(*
Integrates the input error signal with back-calculation anti-windup.

Extends :class:`FB_Integrator` by accepting an external comparator input,
typically the :attr:`~FB_Clamp.Residual` of an :class:`FB_Clamp` block, to
unwind the integrator gradually when the output is saturated. The residual is
scaled by ``1 / Tt`` and subtracted from the integrator input each cycle.

A typical wiring pattern:

.. code-block:: pascal

   fbI.Input           := fbP.Output; // Standard form. Use fError for parallel form.
   fbI.ComparatorInput := fbClamp.Residual;
   fbI.Run();
   fbClamp.Input := fbP.Output + fbI.Output + fbD.Output;
   fbClamp.Run();

.. note::
   Set :attr:`Maximum` before :attr:`Minimum` to ensure the clamp guard applies
   correctly.

   Use ``FB_init`` to set :attr:`tTn` and :attr:`tTt` at declaration time.
*)
{attribute 'no_assign'}
{attribute 'enable_dynamic_creation'}
{attribute 'no_explicit_call' := 'direct call for this function block is not allowed'}
FUNCTION_BLOCK FINAL FB_TrackingIntegrator EXTENDS FB_Integrator
VAR
	_fComparatorInput  : LREAL; // External residual signal for back-calculation anti-windup.
	_tTt 			   : LTIME; // Tracking time constant (Tt). Controls how quickly the integrator unwinds.
END_VAR

(*
Gets or sets the comparator input.

This is typically the :attr:`~FB_Clamp.Residual` of an :class:`FB_Clamp` block
placed after the PID summation, passed directly without negation. The block
subtracts the scaled residual from the integrator input internally to unwind
the integrator when the output is saturated.

A positive value indicates the unsaturated sum exceeded the clamp maximum.
A negative value indicates it fell below the clamp minimum.
*)
PROPERTY ComparatorInput : LREAL
GET
ComparatorInput := THIS^._fComparatorInput;
END_GET
SET
THIS^._fComparatorInput := ComparatorInput;
END_SET
END_PROPERTY

METHOD FB_init : BOOL
VAR_INPUT
	bInitRetains : BOOL;  // if TRUE, the retain variables are initialized (warm start / cold start)
	bInCopyCode  : BOOL;  // if TRUE, the instance afterwards gets moved into the copy code (online change)
	tTn          : LTIME; // Integral action time. LTIME#0 disables integration.
	tTt 		 : LTIME; // Tracking time constant (Tt). A typical starting value is SQRT(Tn * Td).
END_VAR
THIS^._tTt := tTt;
END_METHOD

(*
Advances the tracking integrator by one time step.

.. note::
   Must be called once per cycle on a single PLC task. If :attr:`Tn` is
   ``LTIME#0`` the output is set to zero. If :attr:`Tt` is ``LTIME#0``
   the back-calculation correction is disabled.
*)
METHOD Run
VAR_INST
	{attribute 'hide'}
	bInit       : BOOL := TRUE;
	{attribute 'hide'}
	fT          : LREAL;
	{attribute 'hide'}
	fbTaskCycle : FsCommon.FB_PlcTaskCycleChangeDetector(0);
END_VAR
VAR
	fKi         : LREAL;
	fTt         : LREAL;
	fWindupBack : LREAL;
END_VAR
IF bInit THEN
	fT := TO_LREAL(FsCommon.F_GetCurrentTaskCycleTime()) / TO_LREAL(LTIME#1S);
	RETURN(bInit := fT <= 0);
	fbTaskCycle.TaskIndex := FsCommon.F_GetCurrentTaskIndex();
END_IF

RETURN(NOT fbTaskCycle.HasChanged);

THIS^._fMaximum := MAX(THIS^._fMinimum, THIS^._fMaximum);
THIS^._fMinimum := MIN(THIS^._fMinimum, THIS^._fMaximum);

IF FsCommon.F_ResetOnTrue(THIS^._bSync) THEN
	THIS^._fOutput := LIMIT(THIS^._fMinimum, THIS^._fSync, THIS^._fMaximum);
END_IF

IF THIS^._tTn = LTIME#0S THEN
	THIS^._fOutput := 0;
	RETURN;
END_IF

fKi := 1.0 / (TO_LREAL(THIS^._tTn) / TO_LREAL(LTIME#1S));

IF THIS^._tTt > LTIME#0S THEN
	fTt         := TO_LREAL(THIS^._tTt) / TO_LREAL(LTIME#1S);
	fWindupBack := THIS^._fComparatorInput / fTt;
ELSE
	fWindupBack := 0;
END_IF

THIS^._fOutput := LIMIT(
	THIS^._fMinimum, 
	THIS^._fOutput + (fKi * THIS^._fInput - fWindupBack) * fT,
	THIS^._fMaximum
);
END_METHOD

(*
Gets or sets the tracking time constant (Tt).

Controls how quickly the integrator unwinds after saturation. A typical
starting value is ``SQRT(Tn * Td)``. Setting it to ``LTIME#0`` disables
the back-calculation correction entirely.
*)
PROPERTY Tt : LTIME
GET
Tt := THIS^._tTt;
END_GET
SET
THIS^._tTt := Tt;
END_SET
END_PROPERTY

END_FUNCTION_BLOCK

(* stored: Version 1.1.0.1, ProductVersion 3.1.4024.16
   POU FB_TrackingIntegrator: Id {c82a1daf-bbfa-4a89-a287-ab32f5c04bf6}, SpecialFunc None
   Property ComparatorInput: Id {f18c3236-13f9-4676-a06a-10a11ddd79e4}
   Get Get: Id {243f049c-3d48-40b9-b37f-fdd083fc3b95}
   Set Set: Id {715f49a0-3756-4c2d-b840-4da95b9b1ed2}
   Method FB_init: Id {04699b68-b4a9-4d56-acf6-ad1a410cdcac}
   Method Run: Id {45b7e161-cdeb-4bb4-ba6e-fd45ddcc1b7c}
   Property Tt: Id {ed14ae97-8334-4c39-9c51-575a6eca0eae}
   Get Get: Id {2e4721fc-5d81-4ec9-a4d6-2c1c540d575a}
   Set Set: Id {628f1f72-4e40-4a3c-b188-cdb58589bcd0} *)
